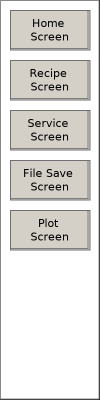
VISUALIZATION vScreenPicker  // 100x400
    Rectangle (0,0 100x400)
    Button (10,10 80x40), "Home Screen"
        OnMouseClick: FrameSelectionChange Selection=Selection=-1, GlobSel=IndExpr=4, AssignDir=vMainScreen.GenElemInst_5, AssignType=Directly, SelType=Globally
    Button (10,60 80x40), "Recipe Screen"
        OnMouseClick: FrameSelectionChange Selection=Selection=-1, GlobSel=IndExpr=1, AssignDir=vMainScreen.GenElemInst_5, AssignType=Directly, SelType=Globally
    Button (10,160 80x40), "File Save Screen"
        OnMouseClick: FrameSelectionChange Selection=Selection=-1, GlobSel=IndExpr=3, AssignDir=vMainScreen.GenElemInst_5, AssignType=Directly, SelType=Globally
    Button (10,110 80x40), "Service Screen"
        OnMouseClick: FrameSelectionChange Selection=Selection=-1, GlobSel=IndExpr=2, AssignDir=vMainScreen.GenElemInst_5, AssignType=Directly, SelType=Globally
    Button (10,210 80x40), "Plot Screen"
        OnMouseClick: FrameSelectionChange Selection=Selection=-1, GlobSel=IndExpr=4, AssignDir=vMainScreen.GenElemInst_5, AssignType=Directly, SelType=Globally
END_VISUALIZATION

(* stored: Version 1.1.0.1, ProductVersion 3.1.4024.12
   Visu vScreenPicker: Id {6d64e162-52a6-4fa1-9908-45a5ce3785db} *)
